(* PLC project Generated.project, CODESYS CODESYS V3.5 SP19 Patch 1 *)
(* stored: creationDateTime 2026-09-06T13:00:42.541781, modificationDateTime 2026-09-06T13:00:42.541781 *)

(* ═══════════════════════════════════════════════════════════════ 🕹️ ST_JoystickChecklist — Diagnostic chronologique communication & prise en main Joystick ─────────────────────────────────────────────────────────────── 🎨 Permet de vérifier la chaîne Joystick (CANopen, Homme-mort, Neutre, Calibration). ═══════════════════════════════════════════════════════════════ *)
TYPE ST_JoystickChecklist : STRUCT
  Step1_CanBusActive : BOOL;  (* 1. Bus & Matériel TRUE = Bus CANopen en état ACTIVE *)
  Step2_JoystickOperational : BOOL;  (* TRUE = Esclave JOY1 en état RUNNING *)
  HwIn_JoyBtnRaw_DI : BOOL;  (* 1bis. Entrées physiques directes HwIn Bouton brut homme-mort issu de HwIn.Operator *)
  NeutralXAct : BOOL;  (* TRUE = Axe X au neutre (PRG_02_Acquisition.Data.Joystick.AxisX.Direction = 0) *)
  NeutralYAct : BOOL;  (* TRUE = Axe Y au neutre (PRG_02_Acquisition.Data.Joystick.AxisY.Direction = 0) *)
  Step3_DeadmanPressed : BOOL;  (* 2. Prise en main & Sécurité TRUE = Bouton Homme-Mort appuyé *)
  Step4_NeutralAcquired : BOOL;  (* TRUE = Repassé par le neutre (autorisation mouvement) *)
  DeadmanArmed : BOOL;  (* TRUE = Homme-Mort armé avec passage au neutre validé *)
  AllConditionsMet : BOOL;  (* 3. Éligibilité globale TRUE = Joystick prêt pour piloter un axe *)
  JoystickSelected : BOOL;  (* TRUE = Joystick maître sélectionné IHM *)
  SelJoystickWinch : INT;  (* Sélection Treuil (0=Couplé M1+M2, 1=M1 seul, 2=M2 seul) *)
  RawX : INT;  (* 4. Mesures brutes & Filtrées Valeur brute axe X (0..10000) *)
  RawY : INT;  (* Valeur brute axe Y (0..10000) *)
  DeflectionX_Pct : REAL;  (* Déflexion signée X (%) *)
  DeflectionY_Pct : REAL;  (* Déflexion signée Y (%) *)
  DirectionX : INT;  (* Direction filtrée X (-1 / 0 / +1) *)
  DirectionY : INT;  (* Direction filtrée Y (-1 / 0 / +1) *)
END_STRUCT;
END_TYPE
